// TIA Portal V19 export
FUNCTION_BLOCK "Area01_SafetyInterface_FB"   // FB66, LAD
TITLE = AREA 01 SAFETY INTERFACE
// stored: Access Published, MemoryReserve 100, SetENOAutomatically false
   VAR_INPUT
      AreaInterface : "AreaInterface";
      Passivation : Bool;
   END_VAR
   VAR_OUTPUT
      MachineInterface : "MachineInterface";
      COut : Struct
         WarningsPresence : Bool;
         AlarmsPresence : Bool;
      END_STRUCT;
   END_VAR
   VAR_IN_OUT
      Alarm : Struct
         FDBACK_Error : Struct
            SafetyValve_CoilCar : Struct
               FDO_FBK_ERROR : Bool;
               EV_SAFETY_FBK_WARNING : Bool;
            END_STRUCT;
            SafetyValve_DecoilersHorizRotation : Struct
               FDO_FBK_ERROR : Bool;
               EV_SAFETY_FBK_WARNING : Bool;
            END_STRUCT;
            SafetyValve_Decoiler1 : Struct
               FDO_FBK_ERROR : Bool;
               EV_SAFETY_FBK_WARNING : Bool;
            END_STRUCT;
            SafetyValve_Decoiler2 : Struct
               FDO_FBK_ERROR : Bool;
               EV_SAFETY_FBK_WARNING : Bool;
            END_STRUCT;
            SafetyValve_Peeler : Struct
               FDO_FBK_ERROR : Bool;
               EV_SAFETY_FBK_WARNING : Bool;
            END_STRUCT;
            SafetyValve_JB_Cut_Rest : Struct
               FDO_FBK_ERROR : Bool;
               EV_SAFETY_FBK_WARNING : Bool;
            END_STRUCT;
            SafetyValve_JB_Cut_Work : Struct
               FDO_FBK_ERROR : Bool;
               EV_SAFETY_FBK_WARNING : Bool;
            END_STRUCT;
            HU_Decoilers_Motor_F_Contactor : Bool;
            HU_Area01_Motor_F_Contactor : Bool;
         END_STRUCT;
         S120_SafetyFaultActive : Struct
            CoilCar : Bool;
            DecoilersTranslation : Bool;
            Decoiler1 : Bool;
            Decoiler2 : Bool;
            Straightener : Bool;
            JBTorch : Bool;
            JBPinchRoll : Bool;
         END_STRUCT;
         UnathorizedOpen : Struct
            D01 : Bool;
            D02 : Bool;
            D03 : Bool;
            D04 : Bool;
            D05 : Bool;
            D07 : Bool;
         END_STRUCT;
      END_STRUCT;
      Warning : Struct
         Selectors : Struct
            Maintenance_MB1 : Bool;
         END_STRUCT;
         DoorOpened : Struct
            D01 : Bool;
            D02 : Bool;
            D03 : Bool;
            D04 : Bool;
            D05 : Bool;
            D06 : Bool;   // NOt EXIST
            D07 : Bool;
         END_STRUCT;
         DoorOpenRequest : Struct
            D01 : Bool;
            D02 : Bool;
            D03 : Bool;
            D04 : Bool;
            D05 : Bool;
            D06 : Bool;   // NOt EXIST
            D07 : Bool;
         END_STRUCT;
         DoorNotLocked : Struct
            D04 : Bool;
            D05 : Bool;
            D07 : Bool;
         END_STRUCT;
      END_STRUCT;
   END_VAR
   VAR
      Sts : Struct
         FdbackErrorPresence : Bool;
         S120SftyFaultPresence : Bool;
         DoorUnauthorizedOpen : Bool;
         DoorOpened { ExternalAccessible := 'False'; ExternalVisible := 'False'; ExternalWritable := 'False'} : Bool;
         DoorOpenRequest : Bool;
         DoorNotLocked : Bool;
      END_STRUCT;
   END_VAR
   VAR_TEMP
      SteadyOn : Bool;
      BlinkFast : Bool;
      BlinkLow : Bool;
      DummyLamp : Bool;
   END_VAR
BEGIN

REGION Network 1: <<<< C O N T R O L S A F E T Y D I A G N O S T I C >>>>>
END_REGION

REGION Network 2 (SCL): Fdback error
   // F FDBACK
   // 
   #Alarm.FDBACK_Error.SafetyValve_CoilCar.FDO_FBK_ERROR := "Main_Safety_RTG1_DB".F_Zone05.F_SafetyValve_CoilCar.FDO_FBK_ERROR;
   #Alarm.FDBACK_Error.SafetyValve_CoilCar.EV_SAFETY_FBK_WARNING := "Main_Safety_RTG1_DB".F_Zone05.F_SafetyValve_CoilCar.EV_SAFETY_FBK_WARNING;


   #Alarm.FDBACK_Error.SafetyValve_DecoilersHorizRotation.FDO_FBK_ERROR := "Main_Safety_RTG1_DB".F_Zone01_02_03.F_SafetyValve_DecoilersHorizRotation.FDO_FBK_ERROR;
   #Alarm.FDBACK_Error.SafetyValve_DecoilersHorizRotation.EV_SAFETY_FBK_WARNING := "Main_Safety_RTG1_DB".F_Zone01_02_03.F_SafetyValve_DecoilersHorizRotation.EV_SAFETY_FBK_WARNING;


   #Alarm.FDBACK_Error.SafetyValve_Decoiler1.FDO_FBK_ERROR := "Main_Safety_RTG1_DB".F_Zone01_02_03.F_SafetyValve_Decoiler1.FDO_FBK_ERROR;
   #Alarm.FDBACK_Error.SafetyValve_Decoiler1.EV_SAFETY_FBK_WARNING := "Main_Safety_RTG1_DB".F_Zone01_02_03.F_SafetyValve_Decoiler1.EV_SAFETY_FBK_WARNING;


   #Alarm.FDBACK_Error.SafetyValve_Decoiler2.FDO_FBK_ERROR := "Main_Safety_RTG1_DB".F_Zone01_02_03.F_SafetyValve_Decoiler2.FDO_FBK_ERROR;
   #Alarm.FDBACK_Error.SafetyValve_Decoiler2.EV_SAFETY_FBK_WARNING := "Main_Safety_RTG1_DB".F_Zone01_02_03.F_SafetyValve_Decoiler2.EV_SAFETY_FBK_WARNING;


   #Alarm.FDBACK_Error.SafetyValve_Peeler.FDO_FBK_ERROR := "Main_Safety_RTG1_DB".F_Zone05.F_SafetyValve_Peeler.FDO_FBK_ERROR;
   #Alarm.FDBACK_Error.SafetyValve_Peeler.EV_SAFETY_FBK_WARNING := "Main_Safety_RTG1_DB".F_Zone05.F_SafetyValve_Peeler.EV_SAFETY_FBK_WARNING;


   #Alarm.FDBACK_Error.SafetyValve_JB_Cut_Rest.FDO_FBK_ERROR := "Main_Safety_RTG1_DB".F_Zone05.F_SafetyValve_JB_Cut_Rest.FDO_FBK_ERROR;
   #Alarm.FDBACK_Error.SafetyValve_JB_Cut_Rest.EV_SAFETY_FBK_WARNING := "Main_Safety_RTG1_DB".F_Zone05.F_SafetyValve_JB_Cut_Rest.EV_SAFETY_FBK_WARNING;


   #Alarm.FDBACK_Error.SafetyValve_JB_Cut_Work.FDO_FBK_ERROR := "Main_Safety_RTG1_DB".F_Zone05.F_SafetyValve_JB_Cut_Work.FDO_FBK_ERROR;
   #Alarm.FDBACK_Error.SafetyValve_JB_Cut_Work.EV_SAFETY_FBK_WARNING := "Main_Safety_RTG1_DB".F_Zone05.F_SafetyValve_JB_Cut_Work.EV_SAFETY_FBK_WARNING;


   #Alarm.FDBACK_Error.HU_Decoilers_Motor_F_Contactor := "Main_Safety_RTG1_DB".F_Zone01_02_03.F_Contactor_HU_Decoilers_Motor.ERROR;
   #Alarm.FDBACK_Error.HU_Area01_Motor_F_Contactor := "Main_Safety_RTG1_DB".F_Zone05.F_Contactor_HU_Area01_Motor.ERROR;
END_REGION

REGION Network 3 (SCL): S120 Safety Fault
   // SINAMICS
   // 
   #Alarm.S120_SafetyFaultActive.CoilCar := "Main_Safety_RTG1_DB".F_Zone00.F_Sinamics_CoilCar.SftyFault;
   #Alarm.S120_SafetyFaultActive.DecoilersTranslation := "Main_Safety_RTG1_DB".F_Zone01_02_03.F_Sinamics_DecoilersTranslation.SftyFault;
   #Alarm.S120_SafetyFaultActive.Decoiler1 := "Main_Safety_RTG1_DB".F_Zone01_02_03.F_Sinamics_Decoiler1.SftyFault;
   #Alarm.S120_SafetyFaultActive.Decoiler2 := "Main_Safety_RTG1_DB".F_Zone01_02_03.F_Sinamics_Decoiler2.SftyFault;
   #Alarm.S120_SafetyFaultActive.Straightener := "Main_Safety_RTG1_DB".F_Zone10.F_Sinamics_Straightener.SftyFault;
   #Alarm.S120_SafetyFaultActive.JBTorch := "Main_Safety_RTG1_DB".F_Zone05.F_Sinamics_JBTorch.SftyFault;
   #Alarm.S120_SafetyFaultActive.JBPinchRoll := "Main_Safety_RTG1_DB".F_Zone05.F_Sinamics_JBPinchRoll.SftyFault;
END_REGION

REGION Network 4: Door D01 - Alarm unauthorized door opening
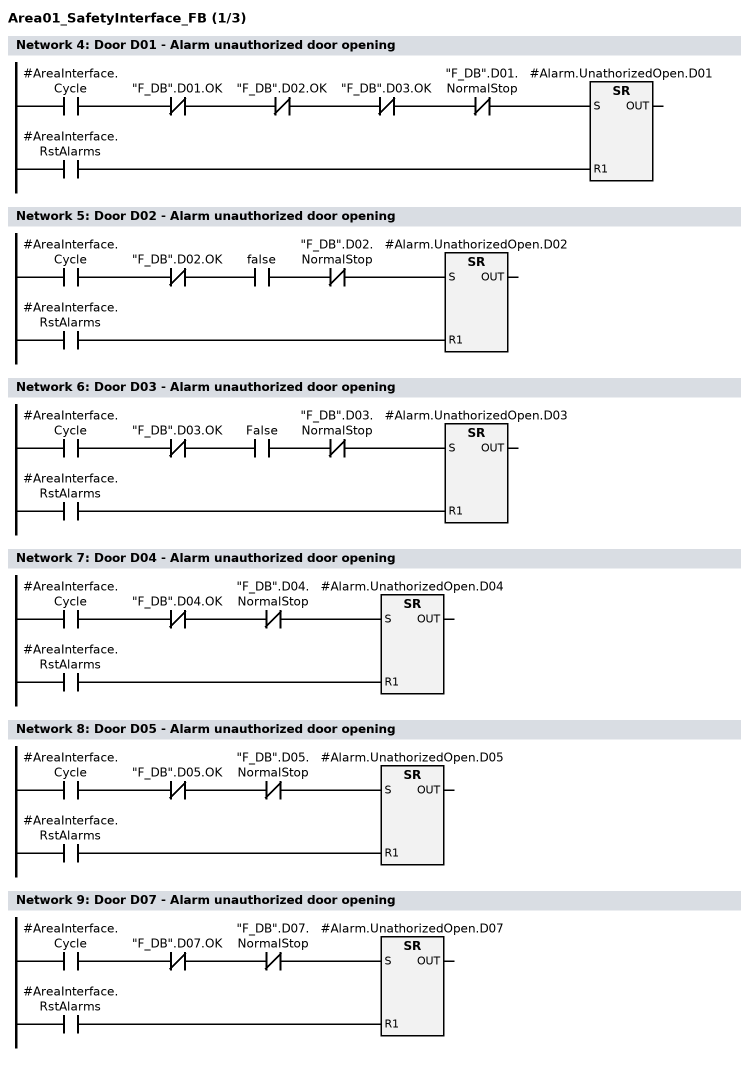
   RUNG wire#powerrail
      Contact( #AreaInterface.Cycle )
      I_Contact( "F_DB".D01.OK )
      I_Contact( "F_DB".D02.OK )
      I_Contact( "F_DB".D03.OK )
      I_Contact( "F_DB".D01.NormalStop )
      S_SR(operand := #Alarm.UnathorizedOpen.D01, r1 := wire#w1)
   END_RUNG
   RUNG wire#powerrail
      Contact( #AreaInterface.RstAlarms )
   END_RUNG wire#w1
   // the same network as SCL:
   IF #AreaInterface.Cycle AND NOT "F_DB".D01.OK AND NOT "F_DB".D02.OK AND NOT "F_DB".D03.OK AND NOT "F_DB".D01.NormalStop THEN
       #Alarm.UnathorizedOpen.D01 := TRUE;   // SR flip-flop
   END_IF;
   IF #AreaInterface.RstAlarms THEN #Alarm.UnathorizedOpen.D01 := FALSE; END_IF;
END_REGION

REGION Network 5: Door D02 - Alarm unauthorized door opening
   RUNG wire#powerrail
      Contact( #AreaInterface.Cycle )
      I_Contact( "F_DB".D02.OK )
      Contact( false )
      I_Contact( "F_DB".D02.NormalStop )
      S_SR(operand := #Alarm.UnathorizedOpen.D02, r1 := wire#w1)
   END_RUNG
   RUNG wire#powerrail
      Contact( #AreaInterface.RstAlarms )
   END_RUNG wire#w1
   // the same network as SCL:
   IF #AreaInterface.Cycle AND NOT "F_DB".D02.OK AND false AND NOT "F_DB".D02.NormalStop THEN
       #Alarm.UnathorizedOpen.D02 := TRUE;   // SR flip-flop
   END_IF;
   IF #AreaInterface.RstAlarms THEN #Alarm.UnathorizedOpen.D02 := FALSE; END_IF;
END_REGION

REGION Network 6: Door D03 - Alarm unauthorized door opening
   RUNG wire#powerrail
      Contact( #AreaInterface.Cycle )
      I_Contact( "F_DB".D03.OK )
      Contact( False )
      I_Contact( "F_DB".D03.NormalStop )
      S_SR(operand := #Alarm.UnathorizedOpen.D03, r1 := wire#w1)
   END_RUNG
   RUNG wire#powerrail
      Contact( #AreaInterface.RstAlarms )
   END_RUNG wire#w1
   // the same network as SCL:
   IF #AreaInterface.Cycle AND NOT "F_DB".D03.OK AND False AND NOT "F_DB".D03.NormalStop THEN
       #Alarm.UnathorizedOpen.D03 := TRUE;   // SR flip-flop
   END_IF;
   IF #AreaInterface.RstAlarms THEN #Alarm.UnathorizedOpen.D03 := FALSE; END_IF;
END_REGION

REGION Network 7: Door D04 - Alarm unauthorized door opening
   RUNG wire#powerrail
      Contact( #AreaInterface.Cycle )
      I_Contact( "F_DB".D04.OK )
      I_Contact( "F_DB".D04.NormalStop )
      S_SR(operand := #Alarm.UnathorizedOpen.D04, r1 := wire#w1)
   END_RUNG
   RUNG wire#powerrail
      Contact( #AreaInterface.RstAlarms )
   END_RUNG wire#w1
   // the same network as SCL:
   IF #AreaInterface.Cycle AND NOT "F_DB".D04.OK AND NOT "F_DB".D04.NormalStop THEN
       #Alarm.UnathorizedOpen.D04 := TRUE;   // SR flip-flop
   END_IF;
   IF #AreaInterface.RstAlarms THEN #Alarm.UnathorizedOpen.D04 := FALSE; END_IF;
END_REGION

REGION Network 8: Door D05 - Alarm unauthorized door opening
   RUNG wire#powerrail
      Contact( #AreaInterface.Cycle )
      I_Contact( "F_DB".D05.OK )
      I_Contact( "F_DB".D05.NormalStop )
      S_SR(operand := #Alarm.UnathorizedOpen.D05, r1 := wire#w1)
   END_RUNG
   RUNG wire#powerrail
      Contact( #AreaInterface.RstAlarms )
   END_RUNG wire#w1
   // the same network as SCL:
   IF #AreaInterface.Cycle AND NOT "F_DB".D05.OK AND NOT "F_DB".D05.NormalStop THEN
       #Alarm.UnathorizedOpen.D05 := TRUE;   // SR flip-flop
   END_IF;
   IF #AreaInterface.RstAlarms THEN #Alarm.UnathorizedOpen.D05 := FALSE; END_IF;
END_REGION

REGION Network 9: Door D07 - Alarm unauthorized door opening
   RUNG wire#powerrail
      Contact( #AreaInterface.Cycle )
      I_Contact( "F_DB".D07.OK )
      I_Contact( "F_DB".D07.NormalStop )
      S_SR(operand := #Alarm.UnathorizedOpen.D07, r1 := wire#w1)
   END_RUNG
   RUNG wire#powerrail
      Contact( #AreaInterface.RstAlarms )
   END_RUNG wire#w1
   // the same network as SCL:
   IF #AreaInterface.Cycle AND NOT "F_DB".D07.OK AND NOT "F_DB".D07.NormalStop THEN
       #Alarm.UnathorizedOpen.D07 := TRUE;   // SR flip-flop
   END_IF;
   IF #AreaInterface.RstAlarms THEN #Alarm.UnathorizedOpen.D07 := FALSE; END_IF;
END_REGION

REGION Network 10: +
END_REGION

REGION Network 11: +
END_REGION

REGION Network 12: +
END_REGION

REGION Network 13: < < < < WARNINGS > > > >
END_REGION

REGION Network 14: Selector set-up MB1
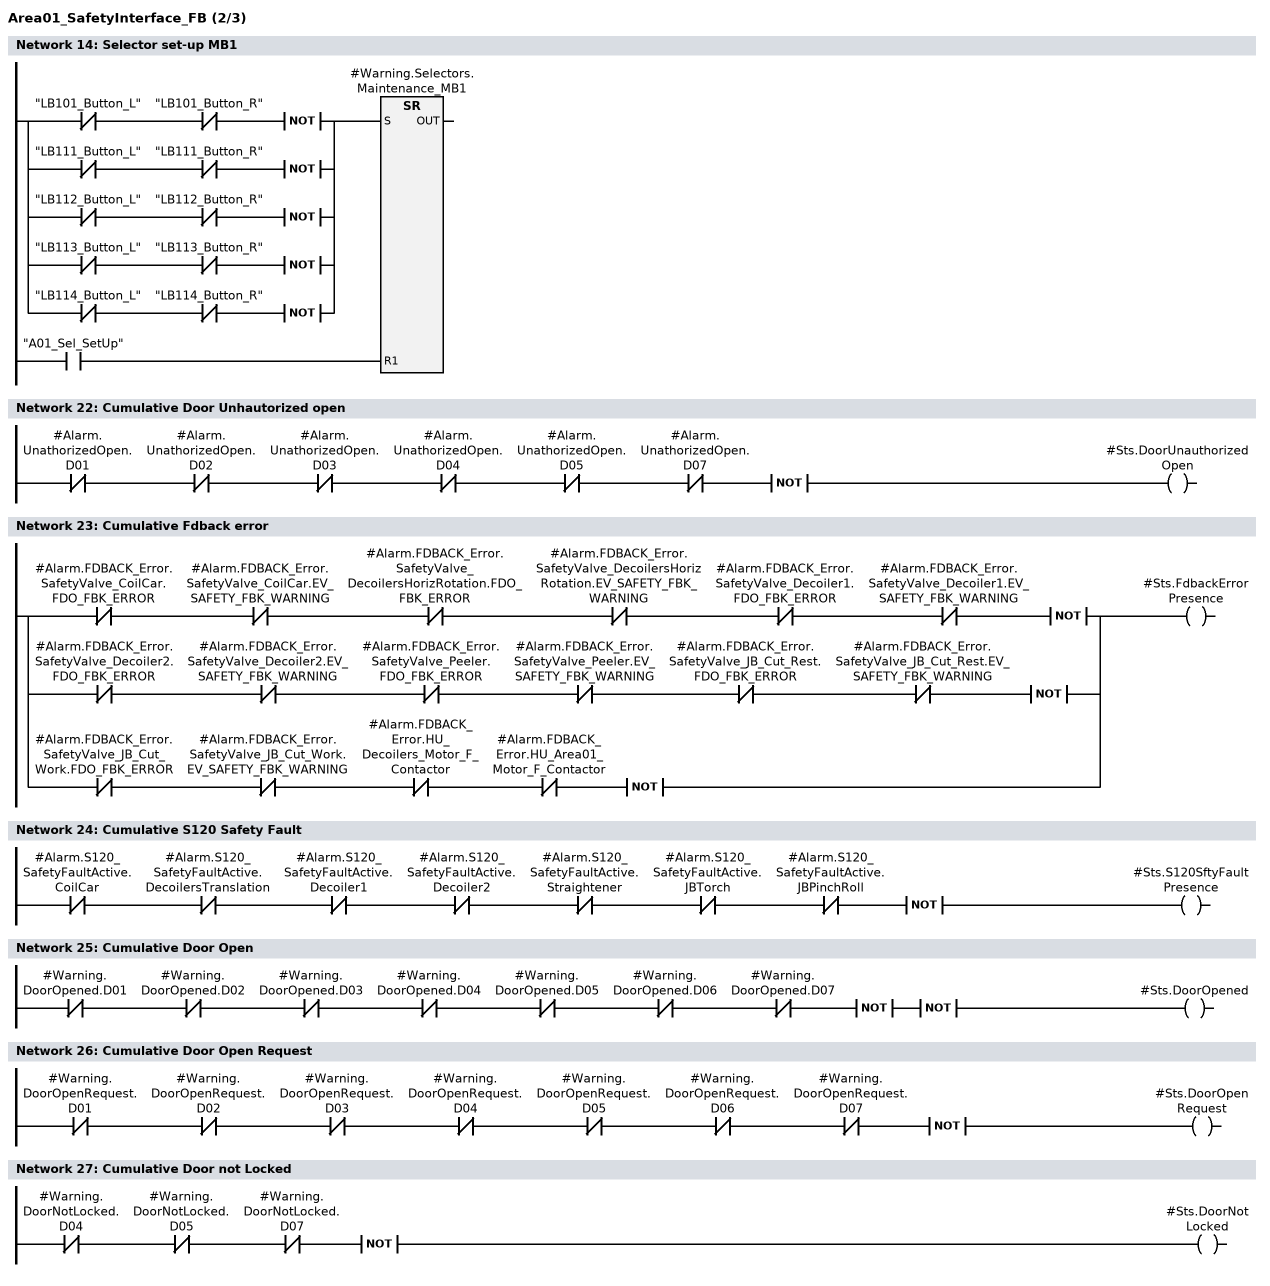
   RUNG wire#powerrail
      I_Contact( "LB101_Button_L" )
      I_Contact( "LB101_Button_R" )
      Not()
      wire#w1
      S_SR(operand := #Warning.Selectors.Maintenance_MB1, r1 := wire#w2)
   END_RUNG
   RUNG wire#powerrail
      I_Contact( "LB111_Button_L" )
      I_Contact( "LB111_Button_R" )
      Not()
   END_RUNG wire#w1
   RUNG wire#powerrail
      I_Contact( "LB112_Button_L" )
      I_Contact( "LB112_Button_R" )
      Not()
   END_RUNG wire#w1
   RUNG wire#powerrail
      I_Contact( "LB113_Button_L" )
      I_Contact( "LB113_Button_R" )
      Not()
   END_RUNG wire#w1
   RUNG wire#powerrail
      I_Contact( "LB114_Button_L" )
      I_Contact( "LB114_Button_R" )
      Not()
   END_RUNG wire#w1
   RUNG wire#powerrail
      Contact( "A01_Sel_SetUp" )
   END_RUNG wire#w2
   // the same network as SCL:
   IF NOT (NOT "LB101_Button_L" AND NOT "LB101_Button_R") OR NOT (NOT "LB111_Button_L" AND NOT "LB111_Button_R") OR NOT (NOT "LB112_Button_L" AND NOT "LB112_Button_R") OR NOT (NOT "LB113_Button_L" AND NOT "LB113_Button_R") OR NOT (NOT "LB114_Button_L" AND NOT "LB114_Button_R") THEN
       #Warning.Selectors.Maintenance_MB1 := TRUE;   // SR flip-flop
   END_IF;
   IF "A01_Sel_SetUp" THEN #Warning.Selectors.Maintenance_MB1 := FALSE; END_IF;
END_REGION

REGION Network 15 (SCL): Door open
   // Door opened
   // 
   #Warning.DoorOpened.D01 := "F_DB".D01.Warning_DoorOpened;
   #Warning.DoorOpened.D02 := "F_DB".D02.Warning_DoorOpened AND "F_DB".D03.Warning_DoorOpened;
   #Warning.DoorOpened.D03 := "F_DB".D03.Warning_DoorOpened AND "F_DB".D02.Warning_DoorOpened;
   #Warning.DoorOpened.D04 := "F_DB".D04.Warning_DoorOpened;
   #Warning.DoorOpened.D05 := "F_DB".D05.Warning_DoorOpened;
   #Warning.DoorOpened.D06 := FALSE;
   #Warning.DoorOpened.D07 := "F_DB".D07.Warning_DoorOpened;
END_REGION

REGION Network 16 (SCL): Door open request
   // Door open reequest
   // 
   #Warning.DoorOpenRequest.D01 := "F_DB".D01.Warning_DoorOpenRequest;
   #Warning.DoorOpenRequest.D02 := "F_DB".D02.Warning_DoorOpenRequest;
   #Warning.DoorOpenRequest.D03 := "F_DB".D03.Warning_DoorOpenRequest;
   #Warning.DoorOpenRequest.D04 := "F_DB".D04.Warning_DoorOpenRequest;
   #Warning.DoorOpenRequest.D05 := "F_DB".D05.Warning_DoorOpenRequest;
   #Warning.DoorOpenRequest.D06 := FALSE;
   #Warning.DoorOpenRequest.D07 := "F_DB".D07.Warning_DoorOpenRequest;
END_REGION

REGION Network 17 (SCL): Door not closed



   #Warning.DoorNotLocked.D04 := "D04_LockEnable" AND NOT "D04_Cancello_Bloccato";
   #Warning.DoorNotLocked.D05 := "D05_LockEnable" AND NOT "D05_Cancello_Bloccato";
   #Warning.DoorNotLocked.D07 := "D07_LockEnable" AND NOT "D07_Cancello_Bloccato";
END_REGION

REGION Network 18: +
END_REGION

REGION Network 19: +
END_REGION

REGION Network 20: +
END_REGION

REGION Network 21: < < < < C U M U L A T I V E > > > >
END_REGION

REGION Network 22: Cumulative Door Unhautorized open
   RUNG wire#powerrail
      I_Contact( #Alarm.UnathorizedOpen.D01 )
      I_Contact( #Alarm.UnathorizedOpen.D02 )
      I_Contact( #Alarm.UnathorizedOpen.D03 )
      I_Contact( #Alarm.UnathorizedOpen.D04 )
      I_Contact( #Alarm.UnathorizedOpen.D05 )
      I_Contact( #Alarm.UnathorizedOpen.D07 )
      Not()
      Coil( #Sts.DoorUnauthorizedOpen )
   END_RUNG
   // the same network as SCL:
   #Sts.DoorUnauthorizedOpen := NOT (NOT #Alarm.UnathorizedOpen.D01 AND NOT #Alarm.UnathorizedOpen.D02 AND NOT #Alarm.UnathorizedOpen.D03 AND NOT #Alarm.UnathorizedOpen.D04 AND NOT #Alarm.UnathorizedOpen.D05 AND NOT #Alarm.UnathorizedOpen.D07);
END_REGION

REGION Network 23: Cumulative Fdback error
   RUNG wire#powerrail
      I_Contact( #Alarm.FDBACK_Error.SafetyValve_CoilCar.FDO_FBK_ERROR )
      I_Contact( #Alarm.FDBACK_Error.SafetyValve_CoilCar.EV_SAFETY_FBK_WARNING )
      I_Contact( #Alarm.FDBACK_Error.SafetyValve_DecoilersHorizRotation.FDO_FBK_ERROR )
      I_Contact( #Alarm.FDBACK_Error.SafetyValve_DecoilersHorizRotation.EV_SAFETY_FBK_WARNING )
      I_Contact( #Alarm.FDBACK_Error.SafetyValve_Decoiler1.FDO_FBK_ERROR )
      I_Contact( #Alarm.FDBACK_Error.SafetyValve_Decoiler1.EV_SAFETY_FBK_WARNING )
      Not()
      wire#w1
      Coil( #Sts.FdbackErrorPresence )
   END_RUNG
   RUNG wire#powerrail
      I_Contact( #Alarm.FDBACK_Error.SafetyValve_Decoiler2.FDO_FBK_ERROR )
      I_Contact( #Alarm.FDBACK_Error.SafetyValve_Decoiler2.EV_SAFETY_FBK_WARNING )
      I_Contact( #Alarm.FDBACK_Error.SafetyValve_Peeler.FDO_FBK_ERROR )
      I_Contact( #Alarm.FDBACK_Error.SafetyValve_Peeler.EV_SAFETY_FBK_WARNING )
      I_Contact( #Alarm.FDBACK_Error.SafetyValve_JB_Cut_Rest.FDO_FBK_ERROR )
      I_Contact( #Alarm.FDBACK_Error.SafetyValve_JB_Cut_Rest.EV_SAFETY_FBK_WARNING )
      Not()
   END_RUNG wire#w1
   RUNG wire#powerrail
      I_Contact( #Alarm.FDBACK_Error.SafetyValve_JB_Cut_Work.FDO_FBK_ERROR )
      I_Contact( #Alarm.FDBACK_Error.SafetyValve_JB_Cut_Work.EV_SAFETY_FBK_WARNING )
      I_Contact( #Alarm.FDBACK_Error.HU_Decoilers_Motor_F_Contactor )
      I_Contact( #Alarm.FDBACK_Error.HU_Area01_Motor_F_Contactor )
      Not()
   END_RUNG wire#w1
   // the same network as SCL:
   #Sts.FdbackErrorPresence := NOT (NOT #Alarm.FDBACK_Error.SafetyValve_CoilCar.FDO_FBK_ERROR AND NOT #Alarm.FDBACK_Error.SafetyValve_CoilCar.EV_SAFETY_FBK_WARNING AND NOT #Alarm.FDBACK_Error.SafetyValve_DecoilersHorizRotation.FDO_FBK_ERROR AND NOT #Alarm.FDBACK_Error.SafetyValve_DecoilersHorizRotation.EV_SAFETY_FBK_WARNING AND NOT #Alarm.FDBACK_Error.SafetyValve_Decoiler1.FDO_FBK_ERROR AND NOT #Alarm.FDBACK_Error.SafetyValve_Decoiler1.EV_SAFETY_FBK_WARNING) OR NOT (NOT #Alarm.FDBACK_Error.SafetyValve_Decoiler2.FDO_FBK_ERROR AND NOT #Alarm.FDBACK_Error.SafetyValve_Decoiler2.EV_SAFETY_FBK_WARNING AND NOT #Alarm.FDBACK_Error.SafetyValve_Peeler.FDO_FBK_ERROR AND NOT #Alarm.FDBACK_Error.SafetyValve_Peeler.EV_SAFETY_FBK_WARNING AND NOT #Alarm.FDBACK_Error.SafetyValve_JB_Cut_Rest.FDO_FBK_ERROR AND NOT #Alarm.FDBACK_Error.SafetyValve_JB_Cut_Rest.EV_SAFETY_FBK_WARNING) OR NOT (NOT #Alarm.FDBACK_Error.SafetyValve_JB_Cut_Work.FDO_FBK_ERROR AND NOT #Alarm.FDBACK_Error.SafetyValve_JB_Cut_Work.EV_SAFETY_FBK_WARNING AND NOT #Alarm.FDBACK_Error.HU_Decoilers_Motor_F_Contactor AND NOT #Alarm.FDBACK_Error.HU_Area01_Motor_F_Contactor);
END_REGION

REGION Network 24: Cumulative S120 Safety Fault
   RUNG wire#powerrail
      I_Contact( #Alarm.S120_SafetyFaultActive.CoilCar )
      I_Contact( #Alarm.S120_SafetyFaultActive.DecoilersTranslation )
      I_Contact( #Alarm.S120_SafetyFaultActive.Decoiler1 )
      I_Contact( #Alarm.S120_SafetyFaultActive.Decoiler2 )
      I_Contact( #Alarm.S120_SafetyFaultActive.Straightener )
      I_Contact( #Alarm.S120_SafetyFaultActive.JBTorch )
      I_Contact( #Alarm.S120_SafetyFaultActive.JBPinchRoll )
      Not()
      Coil( #Sts.S120SftyFaultPresence )
   END_RUNG
   // the same network as SCL:
   #Sts.S120SftyFaultPresence := NOT (NOT #Alarm.S120_SafetyFaultActive.CoilCar AND NOT #Alarm.S120_SafetyFaultActive.DecoilersTranslation AND NOT #Alarm.S120_SafetyFaultActive.Decoiler1 AND NOT #Alarm.S120_SafetyFaultActive.Decoiler2 AND NOT #Alarm.S120_SafetyFaultActive.Straightener AND NOT #Alarm.S120_SafetyFaultActive.JBTorch AND NOT #Alarm.S120_SafetyFaultActive.JBPinchRoll);
END_REGION

REGION Network 25: Cumulative Door Open
   RUNG wire#powerrail
      I_Contact( #Warning.DoorOpened.D01 )
      I_Contact( #Warning.DoorOpened.D02 )
      I_Contact( #Warning.DoorOpened.D03 )
      I_Contact( #Warning.DoorOpened.D04 )
      I_Contact( #Warning.DoorOpened.D05 )
      I_Contact( #Warning.DoorOpened.D06 )
      I_Contact( #Warning.DoorOpened.D07 )
      Not()
      Not()
      Coil( #Sts.DoorOpened )
   END_RUNG
   // the same network as SCL:
   #Sts.DoorOpened := NOT (NOT (NOT #Warning.DoorOpened.D01 AND NOT #Warning.DoorOpened.D02 AND NOT #Warning.DoorOpened.D03 AND NOT #Warning.DoorOpened.D04 AND NOT #Warning.DoorOpened.D05 AND NOT #Warning.DoorOpened.D06 AND NOT #Warning.DoorOpened.D07));
END_REGION

REGION Network 26: Cumulative Door Open Request
   RUNG wire#powerrail
      I_Contact( #Warning.DoorOpenRequest.D01 )
      I_Contact( #Warning.DoorOpenRequest.D02 )
      I_Contact( #Warning.DoorOpenRequest.D03 )
      I_Contact( #Warning.DoorOpenRequest.D04 )
      I_Contact( #Warning.DoorOpenRequest.D05 )
      I_Contact( #Warning.DoorOpenRequest.D06 )
      I_Contact( #Warning.DoorOpenRequest.D07 )
      Not()
      Coil( #Sts.DoorOpenRequest )
   END_RUNG
   // the same network as SCL:
   #Sts.DoorOpenRequest := NOT (NOT #Warning.DoorOpenRequest.D01 AND NOT #Warning.DoorOpenRequest.D02 AND NOT #Warning.DoorOpenRequest.D03 AND NOT #Warning.DoorOpenRequest.D04 AND NOT #Warning.DoorOpenRequest.D05 AND NOT #Warning.DoorOpenRequest.D06 AND NOT #Warning.DoorOpenRequest.D07);
END_REGION

REGION Network 27: Cumulative Door not Locked
   RUNG wire#powerrail
      I_Contact( #Warning.DoorNotLocked.D04 )
      I_Contact( #Warning.DoorNotLocked.D05 )
      I_Contact( #Warning.DoorNotLocked.D07 )
      Not()
      Coil( #Sts.DoorNotLocked )
   END_RUNG
   // the same network as SCL:
   #Sts.DoorNotLocked := NOT (NOT #Warning.DoorNotLocked.D04 AND NOT #Warning.DoorNotLocked.D05 AND NOT #Warning.DoorNotLocked.D07);
END_REGION

REGION Network 28: +
END_REGION

REGION Network 29: +
END_REGION

REGION Network 30: +
END_REGION

REGION Network 31: < < < L A M P S > > >
END_REGION

REGION Network 32: Lamp Safety reset MB1
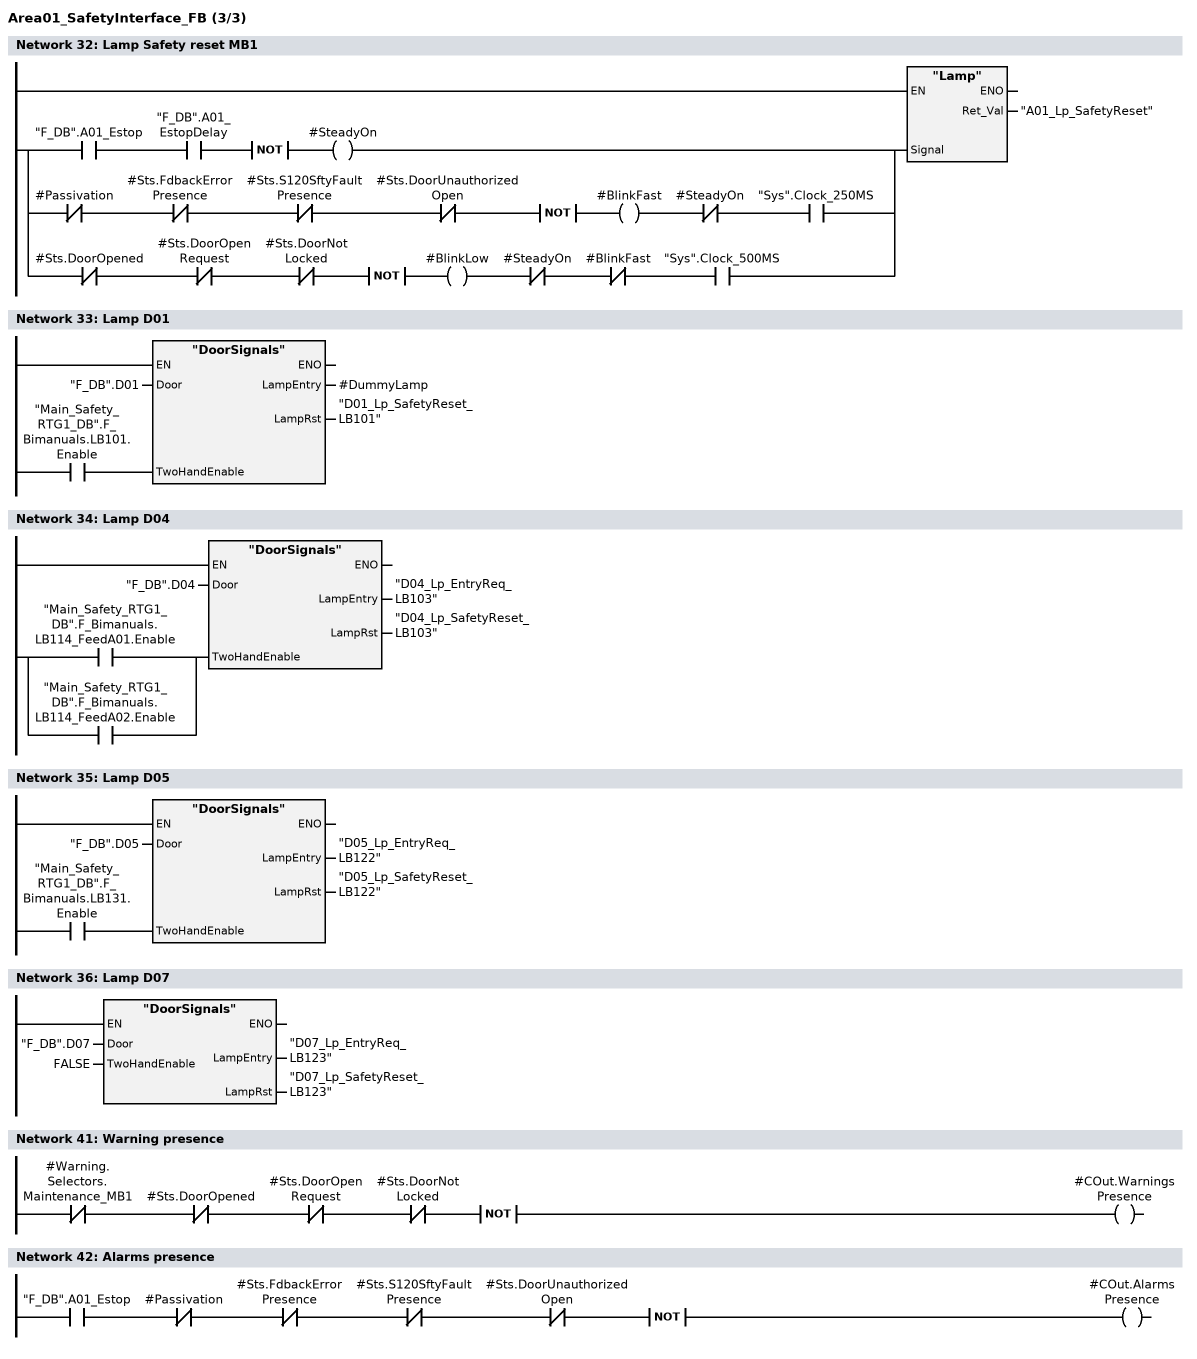
   RUNG wire#powerrail
      "Lamp"(Signal := wire#w1, Ret_Val => "A01_Lp_SafetyReset")
   END_RUNG
   RUNG wire#powerrail
      Contact( "F_DB".A01_Estop )
      Contact( "F_DB".A01_EstopDelay )
      Not()
      Coil( #SteadyOn )
   END_RUNG wire#w1
   RUNG wire#powerrail
      I_Contact( #Passivation )
      I_Contact( #Sts.FdbackErrorPresence )
      I_Contact( #Sts.S120SftyFaultPresence )
      I_Contact( #Sts.DoorUnauthorizedOpen )
      Not()
      Coil( #BlinkFast )
      I_Contact( #SteadyOn )
      Contact( "Sys".Clock_250MS )
   END_RUNG wire#w1
   RUNG wire#powerrail
      I_Contact( #Sts.DoorOpened )
      I_Contact( #Sts.DoorOpenRequest )
      I_Contact( #Sts.DoorNotLocked )
      Not()
      Coil( #BlinkLow )
      I_Contact( #SteadyOn )
      I_Contact( #BlinkFast )
      Contact( "Sys".Clock_500MS )
   END_RUNG wire#w1
   // the same network as SCL:
   #SteadyOn := NOT ("F_DB".A01_Estop AND "F_DB".A01_EstopDelay);
   #BlinkFast := NOT (NOT #Passivation AND NOT #Sts.FdbackErrorPresence AND NOT #Sts.S120SftyFaultPresence AND NOT #Sts.DoorUnauthorizedOpen);
   #BlinkLow := NOT (NOT #Sts.DoorOpened AND NOT #Sts.DoorOpenRequest AND NOT #Sts.DoorNotLocked);
   "A01_Lp_SafetyReset" := "Lamp"(Signal := #SteadyOn OR (#BlinkFast AND NOT #SteadyOn AND "Sys".Clock_250MS) OR (#BlinkLow AND NOT #SteadyOn AND NOT #BlinkFast AND "Sys".Clock_500MS));
END_REGION

REGION Network 33: Lamp D01
   RUNG wire#powerrail
      "DoorSignals"(TwoHandEnable := wire#w1, Door := "F_DB".D01, LampEntry => #DummyLamp, LampRst => "D01_Lp_SafetyReset_LB101")
   END_RUNG
   RUNG wire#powerrail
      Contact( "Main_Safety_RTG1_DB".F_Bimanuals.LB101.Enable )
   END_RUNG wire#w1
   // the same network as SCL:
   "DoorSignals"(Door := "F_DB".D01,
                 TwoHandEnable := "Main_Safety_RTG1_DB".F_Bimanuals.LB101.Enable,
                 LampEntry => #DummyLamp,
                 LampRst => "D01_Lp_SafetyReset_LB101");
END_REGION

REGION Network 34: Lamp D04
   RUNG wire#powerrail
      "DoorSignals"(TwoHandEnable := wire#w1, Door := "F_DB".D04, LampEntry => "D04_Lp_EntryReq_LB103", LampRst => "D04_Lp_SafetyReset_LB103")
   END_RUNG
   RUNG wire#powerrail
      Contact( "Main_Safety_RTG1_DB".F_Bimanuals.LB114_FeedA01.Enable )
   END_RUNG wire#w1
   RUNG wire#powerrail
      Contact( "Main_Safety_RTG1_DB".F_Bimanuals.LB114_FeedA02.Enable )
   END_RUNG wire#w1
   // the same network as SCL:
   "DoorSignals"(Door := "F_DB".D04,
                 TwoHandEnable := "Main_Safety_RTG1_DB".F_Bimanuals.LB114_FeedA01.Enable OR "Main_Safety_RTG1_DB".F_Bimanuals.LB114_FeedA02.Enable,
                 LampEntry => "D04_Lp_EntryReq_LB103",
                 LampRst => "D04_Lp_SafetyReset_LB103");
END_REGION

REGION Network 35: Lamp D05
   RUNG wire#powerrail
      "DoorSignals"(TwoHandEnable := wire#w1, Door := "F_DB".D05, LampEntry => "D05_Lp_EntryReq_LB122", LampRst => "D05_Lp_SafetyReset_LB122")
   END_RUNG
   RUNG wire#powerrail
      Contact( "Main_Safety_RTG1_DB".F_Bimanuals.LB131.Enable )
   END_RUNG wire#w1
   // the same network as SCL:
   "DoorSignals"(Door := "F_DB".D05,
                 TwoHandEnable := "Main_Safety_RTG1_DB".F_Bimanuals.LB131.Enable,
                 LampEntry => "D05_Lp_EntryReq_LB122",
                 LampRst => "D05_Lp_SafetyReset_LB122");
END_REGION

REGION Network 36: Lamp D07
   RUNG wire#powerrail
      "DoorSignals"(Door := "F_DB".D07, TwoHandEnable := FALSE, LampEntry => "D07_Lp_EntryReq_LB123", LampRst => "D07_Lp_SafetyReset_LB123")
   END_RUNG
   // the same network as SCL:
   "DoorSignals"(Door := "F_DB".D07,
                 TwoHandEnable := FALSE,
                 LampEntry => "D07_Lp_EntryReq_LB123",
                 LampRst => "D07_Lp_SafetyReset_LB123");
END_REGION

REGION Network 37: +
END_REGION

REGION Network 38: +
END_REGION

REGION Network 39: +
END_REGION

REGION Network 40: < < < < F I N A L > > > >
END_REGION

REGION Network 41: Warning presence
   RUNG wire#powerrail
      I_Contact( #Warning.Selectors.Maintenance_MB1 )
      I_Contact( #Sts.DoorOpened )
      I_Contact( #Sts.DoorOpenRequest )
      I_Contact( #Sts.DoorNotLocked )
      Not()
      Coil( #COut.WarningsPresence )
   END_RUNG
   // the same network as SCL:
   #COut.WarningsPresence := NOT (NOT #Warning.Selectors.Maintenance_MB1 AND NOT #Sts.DoorOpened AND NOT #Sts.DoorOpenRequest AND NOT #Sts.DoorNotLocked);
END_REGION

REGION Network 42: Alarms presence
   RUNG wire#powerrail
      Contact( "F_DB".A01_Estop )
      I_Contact( #Passivation )
      I_Contact( #Sts.FdbackErrorPresence )
      I_Contact( #Sts.S120SftyFaultPresence )
      I_Contact( #Sts.DoorUnauthorizedOpen )
      Not()
      Coil( #COut.AlarmsPresence )
   END_RUNG
   // the same network as SCL:
   #COut.AlarmsPresence := NOT ("F_DB".A01_Estop AND NOT #Passivation AND NOT #Sts.FdbackErrorPresence AND NOT #Sts.S120SftyFaultPresence AND NOT #Sts.DoorUnauthorizedOpen);
END_REGION

REGION Network 43: >
END_REGION

REGION Network 44: >
END_REGION

REGION Network 45: >
END_REGION

REGION Network 46 (SCL): Collect machine to zone interface

   #MachineInterface.AutReady := #AreaInterface.Aut AND NOT #COut.AlarmsPresence;
   #MachineInterface.Aborting := #COut.AlarmsPresence;
   #MachineInterface.MotionsStandStill := TRUE;
   #MachineInterface.AckStopInPhase := #AreaInterface.StopInPhase;
   #MachineInterface.AckStopProgrammed := #AreaInterface.StopProgrammed;
   #MachineInterface.AlarmsPresence := #COut.AlarmsPresence;
   #MachineInterface.WarningPresence := #COut.WarningsPresence;
END_REGION
END_FUNCTION_BLOCK
